Fanuc KAREL source: IO0093.KL

-- PROVISIONAL review KL for V940-1; original PC SHA256 226081286357804ef59899677bb99a397e902cbf4c20494a26bd1dbd8055439a
-- Incomplete behavior may be omitted. Consult companion uncertainty JSON. Do not deploy.
PROGRAM IO0093
%NOLOCKGROUP
-- UNRESOLVED_LOCAL_POOL 5 cells at code offset 13; source declarations unknown
-- DIRECT_LOCAL_WORD_ACCESS alone does not prove INTEGER, REAL, or BOOLEAN
BEGIN
  -- V9_EXPOSED_INDEXED_TABLE_HINT layout=0001; 1 counted words exposed once; source arms/runtime held
  -- V9_ZERO_GLOBAL_LAYOUT_HINT count-one $GROUP table, zero relocation slots, two routine descriptors; executable preamble and source held
  -- V9_ANALOG_RDI_SIGNAL_HINT AOUT condition array_I
  -- UNRESOLVED_PC offsets 0-18; opcodes 2B,2C,7B
  -- UNRESOLVED_PC offsets 23-30; opcodes 9D,23
  -- UNRESOLVED_PC offsets 35-49; opcodes 2E,22,9D,33,35
  -- UNRESOLVED_PC offsets 54-61; opcodes 9D,23
  -- UNRESOLVED_PC offsets 66-77; opcodes 2E,23
  -- UNRESOLVED_PC offsets 82-105; opcodes 22,21,33,34,19,9C,5B,79
  -- UNRESOLVED_PC offsets 110-124; opcodes 21,9D,52,23
  -- UNRESOLVED_PC offsets 134-138; opcodes 7F
  -- UNRESOLVED_PC offsets 143-147; opcodes 27,AA
  -- UNRESOLVED_PC offsets 152-156; opcodes 7F
END IO0093
